// TIA Portal V20 export
// export: Created 2025-12-01T14:57:25.3928389Z, ExportSetting None, DisplayName Totally Integrated Automation Portal, DisplayVersion V20 Update 3, DisplayName TIA Portal Openness, DisplayVersion V20 Update 3, DisplayName TIA Portal Version Control Interface, DisplayVersion V20 Update 3, DisplayName STEP 7 Professional, DisplayVersion V20 Update 3, DisplayName STEP 7 Safety, DisplayVersion V20 Update 2, DisplayName WinCC Basic/Comfort/Advanced, DisplayVersion V20 Update 3, DisplayName WinCC Professional, DisplayVersion V20 Update 3, DisplayName WinCC Unified, DisplayVersion V20 Update 3
FUNCTION_BLOCK "FB2100_F_CNT_UHS"   // FB2100, F_LAD
{ S7_Optimized_Access := 'TRUE' }
// stored: AutoNumber false
   VAR_INPUT
      IN { ExternalAccessible := 'False'; ExternalVisible := 'False'; ExternalWritable := 'False'} : Bool;   // Contar Tiempo
      R { ExternalAccessible := 'False'; ExternalVisible := 'False'; ExternalWritable := 'False'} : Bool;   // Resetear Tiempo
      PV { ExternalAccessible := 'False'; ExternalVisible := 'False'; ExternalWritable := 'False'} : DInt;   // Valor a Contar (Unidades)
      BaseUnidades_ms : DInt := 100;
   END_VAR
   VAR_OUTPUT
      Q : Bool;
   END_VAR
   VAR
      Valor_Actual { ExternalAccessible := 'False'; ExternalVisible := 'False'; ExternalWritable := 'False'} : DInt;
      Aux_CV { ExternalAccessible := 'False'; ExternalVisible := 'False'; ExternalWritable := 'False'} : DInt;
      STAT_Tiempo_OK { ExternalAccessible := 'False'; ExternalVisible := 'False'; ExternalWritable := 'False'} : Bool;
   END_VAR
   VAR CONSTANT
      CTE_CicloSeguridad : DInt := 50;   // // Tiempo de Interrupción
   END_VAR
BEGIN

REGION Network 1: Inicializar
END_REGION

REGION Network 2: Resetear Tiempo a Cero
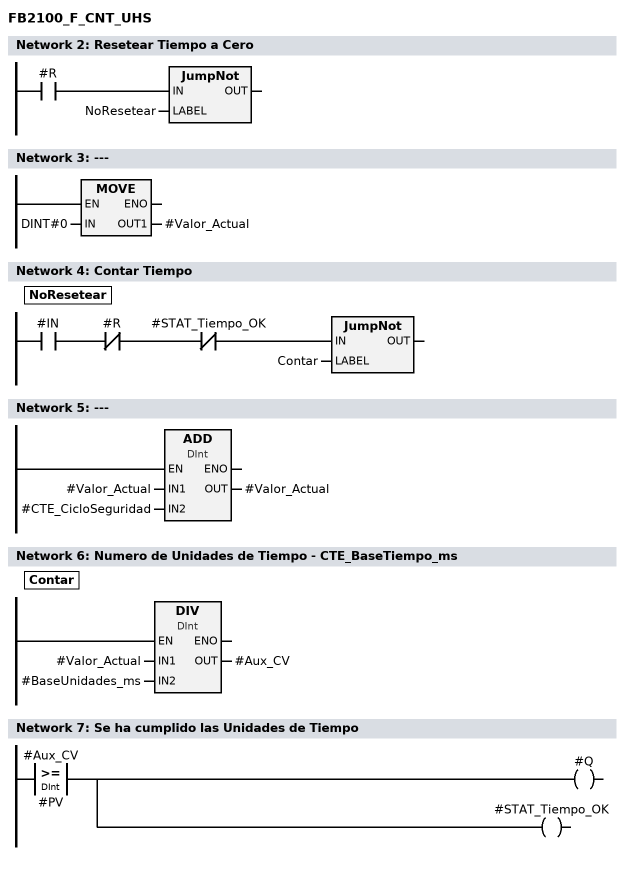
   // no SCL statement known for JumpNot: written as a call
   JumpNot(in := #R, label := NoResetear);
END_REGION

REGION Network 3: ---
   RUNG wire#powerrail
      { S7_GenerateENO := "TRUE" } Move(in := DINT#0, out1 => #Valor_Actual)
   END_RUNG
   // the same network as SCL:
   #Valor_Actual := DINT#0;
END_REGION

REGION Network 4: Contar Tiempo
   // no SCL statement known for JumpNot: written as a call
   NoResetear:
   JumpNot(in := #IN AND NOT #R AND NOT #STAT_Tiempo_OK, label := Contar);
END_REGION

REGION Network 5: ---
   RUNG wire#powerrail
      { S7_Templates := "SrcType := DInt"; S7_GenerateENO := "TRUE" } Add(in1 := #Valor_Actual, in2 := #CTE_CicloSeguridad, out => #Valor_Actual)
   END_RUNG
   // the same network as SCL:
   #Valor_Actual := #Valor_Actual + #CTE_CicloSeguridad;
END_REGION

REGION Network 6: Numero de Unidades de Tiempo - CTE_BaseTiempo_ms
   Label( Contar )
   RUNG wire#powerrail
      { S7_Templates := "SrcType := DInt"; S7_GenerateENO := "TRUE" } Div(in1 := #Valor_Actual, in2 := #BaseUnidades_ms, out => #Aux_CV)
   END_RUNG
   // the same network as SCL:
   Contar:
   #Aux_CV := #Valor_Actual / #BaseUnidades_ms;
END_REGION

REGION Network 7: Se ha cumplido las Unidades de Tiempo
   RUNG wire#powerrail
      { S7_Templates := "SrcType := DInt" } GE_Contact(in1 := #Aux_CV, in2 := #PV)
      wire#w1
      Coil( #Q )
   END_RUNG
   RUNG wire#w1
      Coil( #STAT_Tiempo_OK )
   END_RUNG
   // the same network as SCL:
   #Q := #Aux_CV >= #PV;
   #STAT_Tiempo_OK := #Q;
END_REGION
END_FUNCTION_BLOCK
